{attribute 'GeneratedUsingTerminal: EP3356-0022-0016'}
{attribute addProperty BoxType "EP3356-0022-0016"}
{attribute addProperty Id "StatusAT %I*Status_7BCDA9217"}
{attribute addProperty CRC "3235971242"}
{attribute addProperty Size "7"}
TYPE RMB_Status_C0E100AA :
STRUCT
	{attribute addProperty Name "Status"}
	Status AT %I* : Status_7BCDA921;
END_STRUCT
END_TYPE

(* stored: Version 1.2.0.0, ProductVersion 3.1.4024.9
   DUT RMB_Status_C0E100AA: Id {560e7cc1-d41b-4982-a8cd-e9ef727b9c1e} *)
